// TIA Portal V18 export
DATA_BLOCK "Potlife"   // DB73
{ S7_Optimized_Access := 'TRUE' }
VERSION : 0.1
// stored: AutoNumber true, DBAccessibleFromOPCUA true, IsOnlyStoredInLoadMemory false, IsRetainMemResEnabled false, IsWriteProtectedInAS false, MemoryReserve 100
   VAR
      "run time" : Struct
         Hours : Int := 0;
         minutes : Int := 0;
         seconds : Int := 0;
      END_STRUCT;
   END_VAR
   VAR RETAIN
      "set time format" : Int := 0;
      "enable potlife" : Int := 0;
   END_VAR
   VAR
      "potlife life enabled" : Bool := FALSE;
   END_VAR
   VAR RETAIN
      "set time" : Int := 30;
   END_VAR
   VAR
      "Potlife time in seconds" : Bool := FALSE;
      "potlife time in minutes" : Bool := TRUE;
   END_VAR
   VAR RETAIN
      "Mixing Volume to dispense" : Real := 3.0;
      Flowrate : Real := 3.0;
      "Control time" : Int := 60;
   END_VAR
   VAR
      "Control time in sec" : DInt := -5536;
   END_VAR
   VAR RETAIN
      "Maximum number of cycle" : Int := 5;
   END_VAR
   VAR
      "potlifetime format" : Int := 0;
      "set time input" : Struct
         seconds : DInt := 30000;
         minutes : DInt := 1800000;
      END_STRUCT;
      contol : Struct
         "trigger potlife" : Bool := TRUE;
         "Potlife elapsed Start Regeneration" : Bool := TRUE;
         "start potlife timer" : Bool := TRUE;
         "Seconds timer Done" : Bool := FALSE;
         "minutes timer Done" : Bool := TRUE;
         "60sec pulse done" : Bool := FALSE;
         "reset counter" : Bool := TRUE;
         "Potlife elapsed machine not in regeneration" : Bool := TRUE;
         "start reneration program" : Bool := FALSE;
         "Start Sequence" : Bool := FALSE;
      END_STRUCT;
      "Time PV" : Struct
         "Sectimer PV" : DInt := 0;
         minutestimerPV : DInt := 1800000;
         "secPulse PV" : Int := 0;
      END_STRUCT;
      "Time PV unscalled" : Struct
         "Sectimer PV" : Int := 0;
         minutestimerPV : Int := 30;
         "secPulse PV" : Int := 0;
      END_STRUCT;
      "Time PV Down Counts" : Struct
         "Sectimer PV" : DInt := 0;
         minutestimerPV : DInt := 0;
         "secPulse PV" : Int := 0;
      END_STRUCT;
      "Flush Control" : Struct
         "maximum cycle reached" : Bool := FALSE;
         "Flush pgm selected" : Bool := FALSE;
         "start Flush" : Bool := FALSE;
      END_STRUCT;
      "Control time in sec_1" : DInt;
   END_VAR
BEGIN
END_DATA_BLOCK
